// Mitsubishi GX Works2 project: EX2 (3)   PLC: FX3G

// global labels: Global1
VAR_GLOBAL
  Emergency AT X005 : BOOL;
  End_Day AT M1 : BOOL;
  Start_Day AT X007 : BOOL;
  Work_Active AT M0 : BOOL;
  Work_Light AT Y007 : BOOL;
  No_Stock AT M6 : BOOL;
  Start_Process AT X001 : BOOL;
  Analog_Input_1 AT D8280 : INT;
  Sample_Done AT M2 : BOOL;
  Regular_Type AT M3 : BOOL;
  Premium_Type AT M4 : BOOL;
  Reg_Raspberry_OK AT M20 : BOOL;
  Reg_Lemon_OK AT M21 : BOOL;
  Reg_Stabilizer_OK AT M22 : BOOL;
  Reg_Gummies_OK AT M23 : BOOL;
  Regular_Stock_OK AT M14 : BOOL;
  Prem_Raspberry_OK AT M24 : BOOL;
  Prem_Lemon_OK AT M25 : BOOL;
  Prem_Stabilizer_OK AT M26 : BOOL;
  Prem_Gummies_OK AT M27 : BOOL;
  Premium_Stock_OK AT M15 : BOOL;
  Stock_OK AT M5 : BOOL;
  Prep_Active AT M7 : BOOL;
  Prep_Timer AT TC0 : BOOL;
  Prep_Timer_Done AT TS0 : BOOL;
  Prep_Light AT Y000 : BOOL;
  Prep_Done AT M8 : BOOL;
  Start_Cooling AT X002 : BOOL;
  Cooling_Active AT M9 : BOOL;
  Cooling_Timer AT TC1 : BOOL;
  Cooling_done AT M10 : BOOL;
  Cooling_Light AT Y002 : BOOL;
  Cooling_Timer_Done AT TS1 : BOOL;
  Temp_Sensor AT X003 : BOOL;
  Mixing_Active AT M11 : BOOL;
  Mixing_Timer_Reg AT TC2 : BOOL;
  Mixing_Timer_Prem AT TC3 : BOOL;
  Blink_Timer_Done_2 AT TS5 : BOOL;
  Blink_Timer_2_Done AT TS5 : BOOL;
  Blink_Timer_1 AT TC4 : BOOL;
  Blink_Timer_1_Done AT TS4 : BOOL;
  Blink_Timer_2 AT TC5 : BOOL;
  Mixing_Light_1 AT Y005 : BOOL;
  Mixing_Light_2 AT Y006 : BOOL;
  Blink_Light_1 AT Y005 : BOOL;
  Blink_Light_2 AT Y006 : BOOL;
  Mixing_Timer_Reg_Done AT TS2 : BOOL;
  Mixing_Timer_Prem_Done AT TS3 : BOOL;
  Mixing_Done AT M12 : BOOL;
END_VAR
VAR_GLOBAL CONSTANT
  One_Package : REAL := 1.0;
END_VAR
VAR_GLOBAL
  Cycle_Reset AT M13 : BOOL;
END_VAR
VAR_GLOBAL CONSTANT
  Ten : REAL;
END_VAR
VAR_GLOBAL
  Analog_Display_Value AT D1280 : REAL;
  Analog_Output AT D8282 : INT;
  Zero AT D0 : REAL;
  Analog_Value AT D1100 : REAL;
END_VAR
VAR_GLOBAL CONSTANT
  Regular_Max : REAL;
  Premium_Min : REAL;
END_VAR
VAR_GLOBAL
  Raspberry_Stock AT D1110 : REAL;
  Reg_Raspberry_Need AT D1190 : REAL;
  Lemon_Stock AT D1120 : REAL;
  Reg_Lemon_Need AT D1200 : REAL;
  Gummies_Stock AT D1140 : REAL;
  Prem_Raspberry_Need AT D1230 : REAL;
  Prem_Lemon_Need AT D1240 : REAL;
  Storage_Count AT D1270 : REAL;
  Reg_Gummies_Need AT D1220 : REAL;
  Prem_Gummies_Need AT D1260 : REAL;
  Reg_Stabilizer_Need AT D1210 : REAL;
  Stabilizer_Stock AT D1130 : REAL;
  Prem_Stabilizer_Need AT D1250 : REAL;
  Raspberry_Need AT D1190 : REAL;
  Lemon_Need AT D1200 : REAL;
  Gummies_Need AT D1220 : REAL;
  Stabilizer_Need AT D1210 : REAL;
  Raspberry_OK AT M20 : BOOL;
  Lemon_OK AT M21 : BOOL;
  Stabilizer_OK AT M22 : BOOL;
  Gummies_OK AT M23 : BOOL;
  Input_Raspberry_Stock AT D1500 : REAL;
  Input_Lemon_Stock AT D1510 : REAL;
  Input_Stabilizer_Stock AT D1520 : REAL;
  Input_Gummies_Stock AT D1530 : REAL;
  Raspberry_Cooling_Tank AT D1300 : REAL;
  Lemon_Cooling_Tank AT D1310 : REAL;
  Mixing_Tank AT D1320 : REAL;
  Not_valid_value AT M28 : BOOL;
  Premium_Min_Check AT M29 : BOOL;
  Premium_Max_Check AT M30 : BOOL;
  Invalid_Min_Check AT M31 : BOOL;
  Invalid_Max_Check AT M32 : BOOL;
  Invalid_Range_Check AT M33 : BOOL;
  Above_10_Check AT M34 : BOOL;
END_VAR
VAR_GLOBAL CONSTANT
  Con2400 : REAL := 2400;
  Con4000 : REAL := 4000.0;
  Con_40 : REAL := 40.0;
END_VAR
VAR_GLOBAL
  Storage_multi_40 AT D1290 : REAL;
END_VAR
VAR_GLOBAL CONSTANT
  Con_210 : REAL := 210.0;
END_VAR

// task Task_01 (event TRUE, interval 0, priority 31): POU_01

PROGRAM POU_01
(* structured ladder/FBD written out as ST: instructions are called as NAME(EN, inputs, outputs); _pN, _eN, _tN stand for wires *)
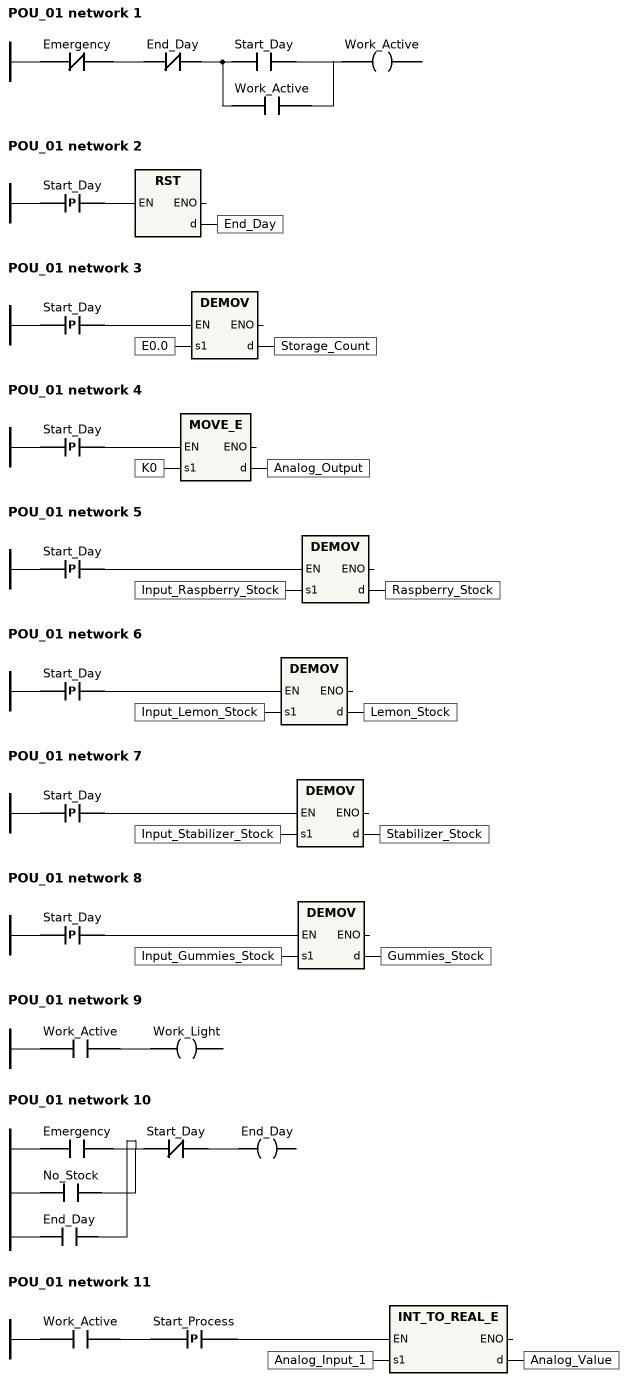
(* network 1 *)
_p1 := NOT Emergency AND NOT End_Day;
Work_Active := (_p1 AND Start_Day) OR (_p1 AND Work_Active);
(* network 2 *)
RST(LDP(TRUE, Start_Day), End_Day);
(* network 3 *)
DEMOV(LDP(TRUE, Start_Day), E0.0, Storage_Count);
(* network 4 *)
MOVE_E(LDP(TRUE, Start_Day), K0, Analog_Output);
(* network 5 *)
DEMOV(LDP(TRUE, Start_Day), Input_Raspberry_Stock, Raspberry_Stock);
(* network 6 *)
DEMOV(LDP(TRUE, Start_Day), Input_Lemon_Stock, Lemon_Stock);
(* network 7 *)
DEMOV(LDP(TRUE, Start_Day), Input_Stabilizer_Stock, Stabilizer_Stock);
(* network 8 *)
DEMOV(LDP(TRUE, Start_Day), Input_Gummies_Stock, Gummies_Stock);
(* network 9 *)
Work_Light := Work_Active;
(* network 10 *)
End_Day := (Emergency OR No_Stock OR End_Day) AND NOT Start_Day;
(* network 11 *)
INT_TO_REAL_E(Work_Active AND LDP(TRUE, Start_Process), Analog_Input_1, Analog_Value);
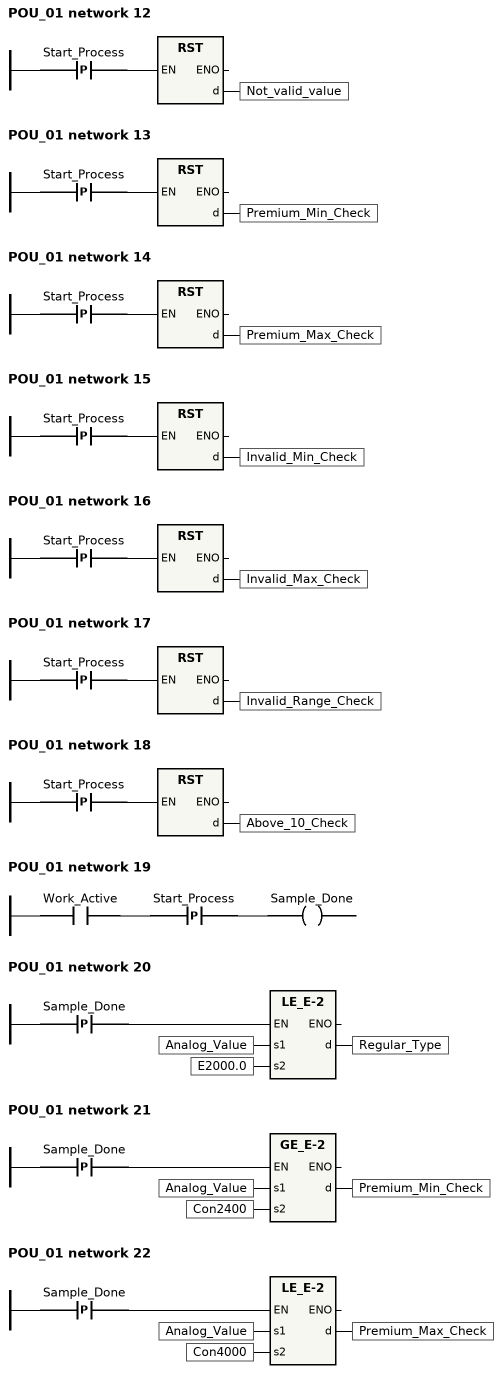
(* network 12 *)
RST(LDP(TRUE, Start_Process), Not_valid_value);
(* network 13 *)
RST(LDP(TRUE, Start_Process), Premium_Min_Check);
(* network 14 *)
RST(LDP(TRUE, Start_Process), Premium_Max_Check);
(* network 15 *)
RST(LDP(TRUE, Start_Process), Invalid_Min_Check);
(* network 16 *)
RST(LDP(TRUE, Start_Process), Invalid_Max_Check);
(* network 17 *)
RST(LDP(TRUE, Start_Process), Invalid_Range_Check);
(* network 18 *)
RST(LDP(TRUE, Start_Process), Above_10_Check);
(* network 19 *)
Sample_Done := Work_Active AND LDP(TRUE, Start_Process);
(* network 20 *)
LE_E(LDP(TRUE, Sample_Done), Analog_Value, E2000.0, Regular_Type);
(* network 21 *)
GE_E(LDP(TRUE, Sample_Done), Analog_Value, Con2400, Premium_Min_Check);
(* network 22 *)
LE_E(LDP(TRUE, Sample_Done), Analog_Value, Con4000, Premium_Max_Check);
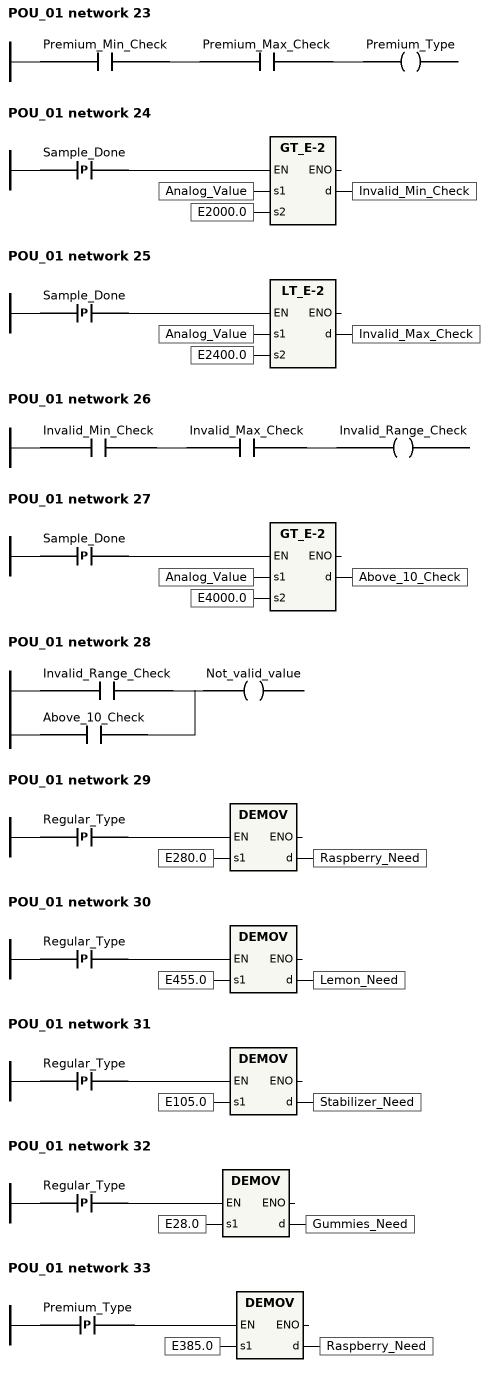
(* network 23 *)
Premium_Type := Premium_Min_Check AND Premium_Max_Check;
(* network 24 *)
GT_E(LDP(TRUE, Sample_Done), Analog_Value, E2000.0, Invalid_Min_Check);
(* network 25 *)
LT_E(LDP(TRUE, Sample_Done), Analog_Value, E2400.0, Invalid_Max_Check);
(* network 26 *)
Invalid_Range_Check := Invalid_Min_Check AND Invalid_Max_Check;
(* network 27 *)
GT_E(LDP(TRUE, Sample_Done), Analog_Value, E4000.0, Above_10_Check);
(* network 28 *)
Not_valid_value := Invalid_Range_Check OR Above_10_Check;
(* network 29 *)
DEMOV(LDP(TRUE, Regular_Type), E280.0, Raspberry_Need);
(* network 30 *)
DEMOV(LDP(TRUE, Regular_Type), E455.0, Lemon_Need);
(* network 31 *)
DEMOV(LDP(TRUE, Regular_Type), E105.0, Stabilizer_Need);
(* network 32 *)
DEMOV(LDP(TRUE, Regular_Type), E28.0, Gummies_Need);
(* network 33 *)
DEMOV(LDP(TRUE, Premium_Type), E385.0, Raspberry_Need);
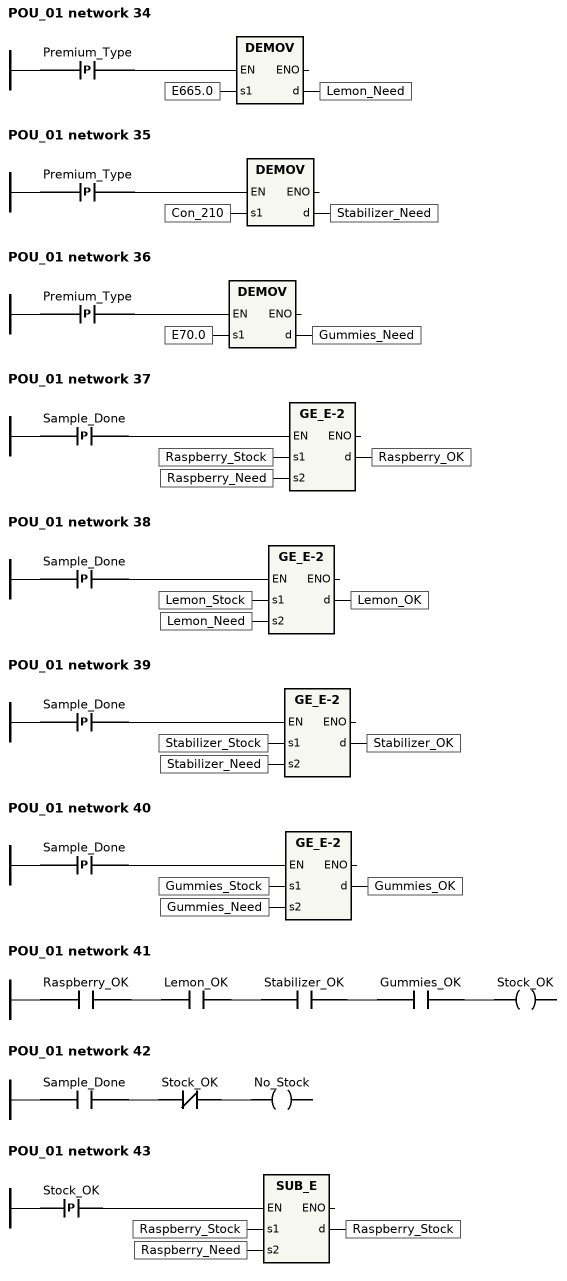
(* network 34 *)
DEMOV(LDP(TRUE, Premium_Type), E665.0, Lemon_Need);
(* network 35 *)
DEMOV(LDP(TRUE, Premium_Type), Con_210, Stabilizer_Need);
(* network 36 *)
DEMOV(LDP(TRUE, Premium_Type), E70.0, Gummies_Need);
(* network 37 *)
GE_E(LDP(TRUE, Sample_Done), Raspberry_Stock, Raspberry_Need, Raspberry_OK);
(* network 38 *)
GE_E(LDP(TRUE, Sample_Done), Lemon_Stock, Lemon_Need, Lemon_OK);
(* network 39 *)
GE_E(LDP(TRUE, Sample_Done), Stabilizer_Stock, Stabilizer_Need, Stabilizer_OK);
(* network 40 *)
GE_E(LDP(TRUE, Sample_Done), Gummies_Stock, Gummies_Need, Gummies_OK);
(* network 41 *)
Stock_OK := Raspberry_OK AND Lemon_OK AND Stabilizer_OK AND Gummies_OK;
(* network 42 *)
No_Stock := Sample_Done AND NOT Stock_OK;
(* network 43 *)
SUB_E(LDP(TRUE, Stock_OK), Raspberry_Stock, Raspberry_Need, Raspberry_Stock);
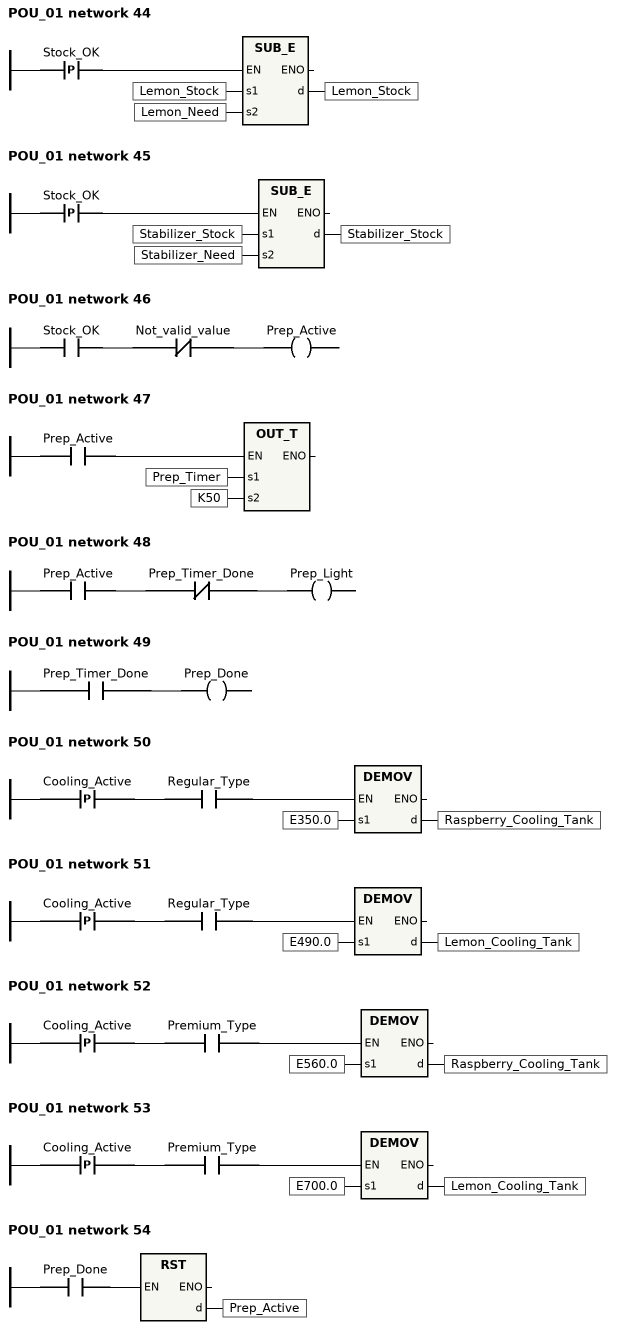
(* network 44 *)
SUB_E(LDP(TRUE, Stock_OK), Lemon_Stock, Lemon_Need, Lemon_Stock);
(* network 45 *)
SUB_E(LDP(TRUE, Stock_OK), Stabilizer_Stock, Stabilizer_Need, Stabilizer_Stock);
(* network 46 *)
Prep_Active := Stock_OK AND NOT Not_valid_value;
(* network 47 *)
OUT_T(Prep_Active, Prep_Timer, K50);
(* network 48 *)
Prep_Light := Prep_Active AND NOT Prep_Timer_Done;
(* network 49 *)
Prep_Done := Prep_Timer_Done;
(* network 50 *)
DEMOV(LDP(TRUE, Cooling_Active) AND Regular_Type, E350.0, Raspberry_Cooling_Tank);
(* network 51 *)
DEMOV(LDP(TRUE, Cooling_Active) AND Regular_Type, E490.0, Lemon_Cooling_Tank);
(* network 52 *)
DEMOV(LDP(TRUE, Cooling_Active) AND Premium_Type, E560.0, Raspberry_Cooling_Tank);
(* network 53 *)
DEMOV(LDP(TRUE, Cooling_Active) AND Premium_Type, E700.0, Lemon_Cooling_Tank);
(* network 54 *)
RST(Prep_Done, Prep_Active);
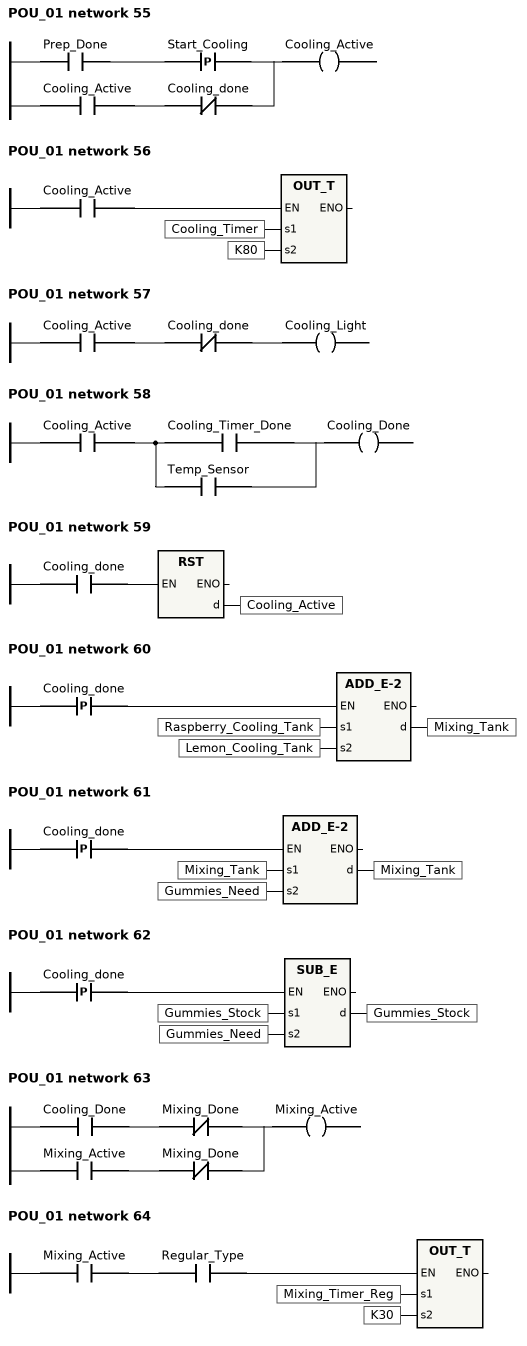
(* network 55 *)
Cooling_Active := (Prep_Done AND LDP(TRUE, Start_Cooling)) OR (Cooling_Active AND NOT Cooling_done);
(* network 56 *)
OUT_T(Cooling_Active, Cooling_Timer, K80);
(* network 57 *)
Cooling_Light := Cooling_Active AND NOT Cooling_done;
(* network 58 *)
Cooling_Done := (Cooling_Active AND Cooling_Timer_Done) OR (Cooling_Active AND Temp_Sensor);
(* network 59 *)
RST(Cooling_done, Cooling_Active);
(* network 60 *)
ADD_E(LDP(TRUE, Cooling_done), Raspberry_Cooling_Tank, Lemon_Cooling_Tank, Mixing_Tank);
(* network 61 *)
ADD_E(LDP(TRUE, Cooling_done), Mixing_Tank, Gummies_Need, Mixing_Tank);
(* network 62 *)
SUB_E(LDP(TRUE, Cooling_done), Gummies_Stock, Gummies_Need, Gummies_Stock);
(* network 63 *)
Mixing_Active := (Cooling_Done AND NOT Mixing_Done) OR (Mixing_Active AND NOT Mixing_Done);
(* network 64 *)
OUT_T(Mixing_Active AND Regular_Type, Mixing_Timer_Reg, K30);
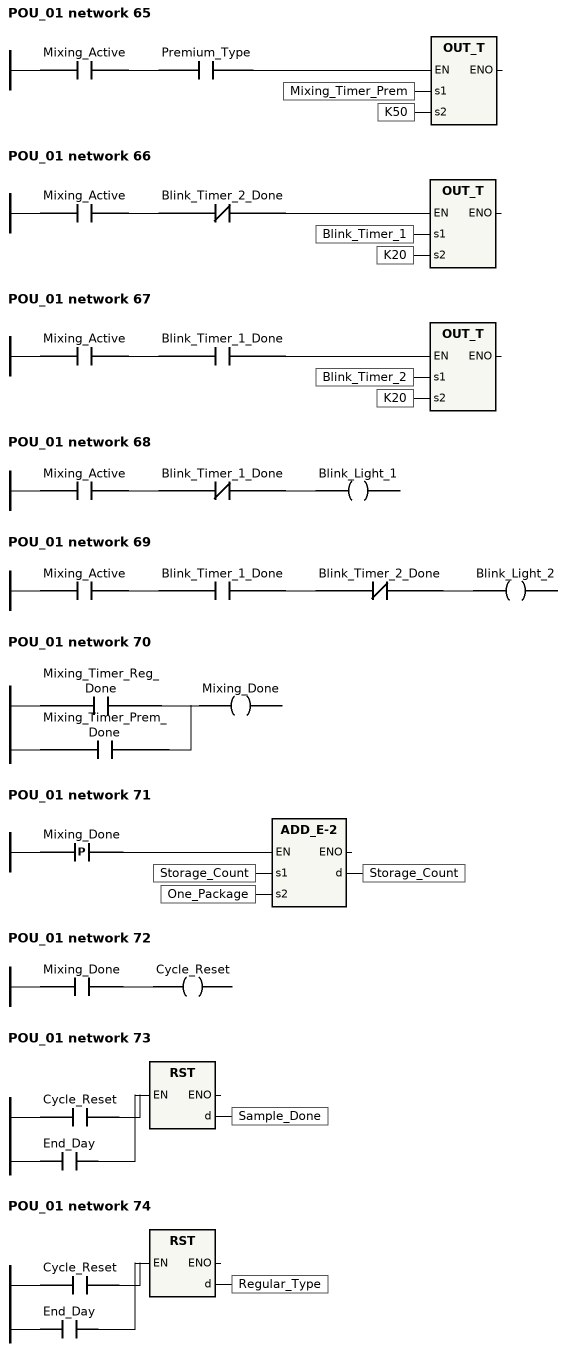
(* network 65 *)
OUT_T(Mixing_Active AND Premium_Type, Mixing_Timer_Prem, K50);
(* network 66 *)
OUT_T(Mixing_Active AND NOT Blink_Timer_2_Done, Blink_Timer_1, K20);
(* network 67 *)
OUT_T(Mixing_Active AND Blink_Timer_1_Done, Blink_Timer_2, K20);
(* network 68 *)
Blink_Light_1 := Mixing_Active AND NOT Blink_Timer_1_Done;
(* network 69 *)
Blink_Light_2 := Mixing_Active AND Blink_Timer_1_Done AND NOT Blink_Timer_2_Done;
(* network 70 *)
Mixing_Done := Mixing_Timer_Reg_Done OR Mixing_Timer_Prem_Done;
(* network 71 *)
ADD_E(LDP(TRUE, Mixing_Done), Storage_Count, One_Package, Storage_Count);
(* network 72 *)
Cycle_Reset := Mixing_Done;
(* network 73 *)
RST(Cycle_Reset OR End_Day, Sample_Done);
(* network 74 *)
RST(Cycle_Reset OR End_Day, Regular_Type);
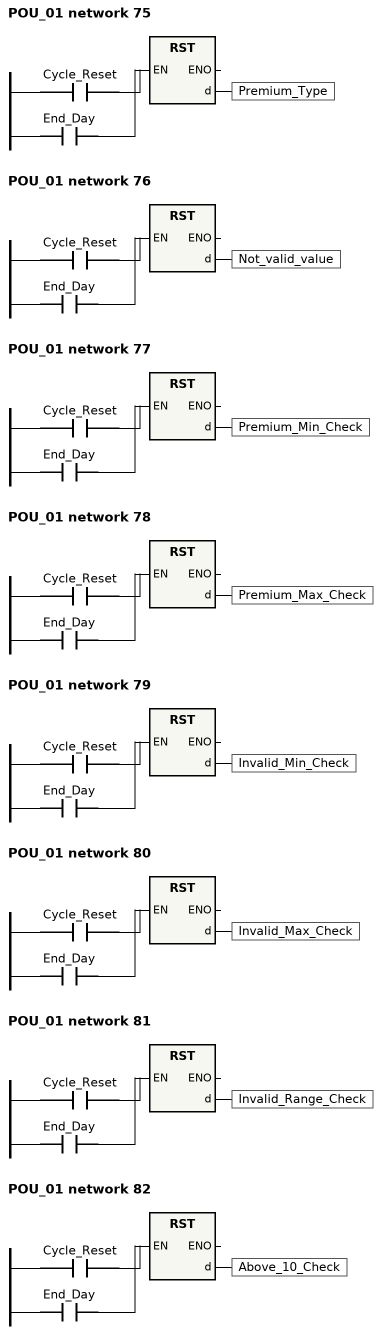
(* network 75 *)
RST(Cycle_Reset OR End_Day, Premium_Type);
(* network 76 *)
RST(Cycle_Reset OR End_Day, Not_valid_value);
(* network 77 *)
RST(Cycle_Reset OR End_Day, Premium_Min_Check);
(* network 78 *)
RST(Cycle_Reset OR End_Day, Premium_Max_Check);
(* network 79 *)
RST(Cycle_Reset OR End_Day, Invalid_Min_Check);
(* network 80 *)
RST(Cycle_Reset OR End_Day, Invalid_Max_Check);
(* network 81 *)
RST(Cycle_Reset OR End_Day, Invalid_Range_Check);
(* network 82 *)
RST(Cycle_Reset OR End_Day, Above_10_Check);
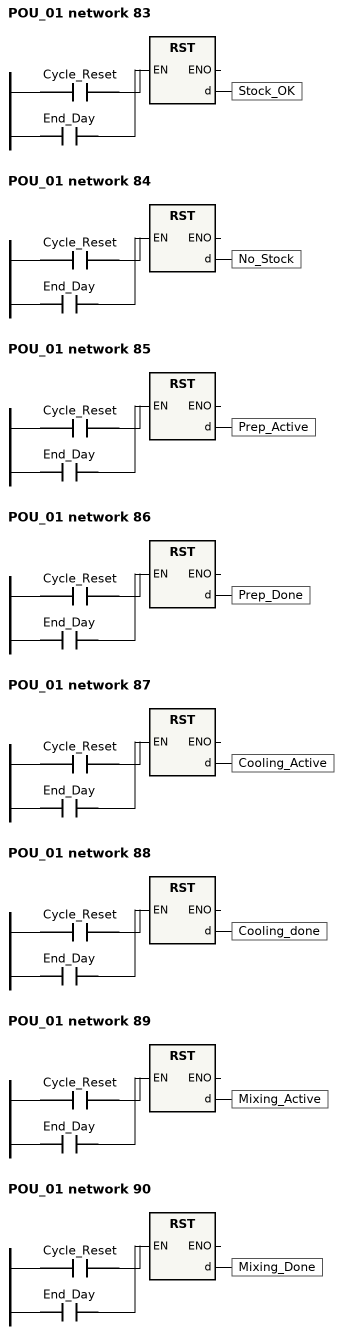
(* network 83 *)
RST(Cycle_Reset OR End_Day, Stock_OK);
(* network 84 *)
RST(Cycle_Reset OR End_Day, No_Stock);
(* network 85 *)
RST(Cycle_Reset OR End_Day, Prep_Active);
(* network 86 *)
RST(Cycle_Reset OR End_Day, Prep_Done);
(* network 87 *)
RST(Cycle_Reset OR End_Day, Cooling_Active);
(* network 88 *)
RST(Cycle_Reset OR End_Day, Cooling_done);
(* network 89 *)
RST(Cycle_Reset OR End_Day, Mixing_Active);
(* network 90 *)
RST(Cycle_Reset OR End_Day, Mixing_Done);
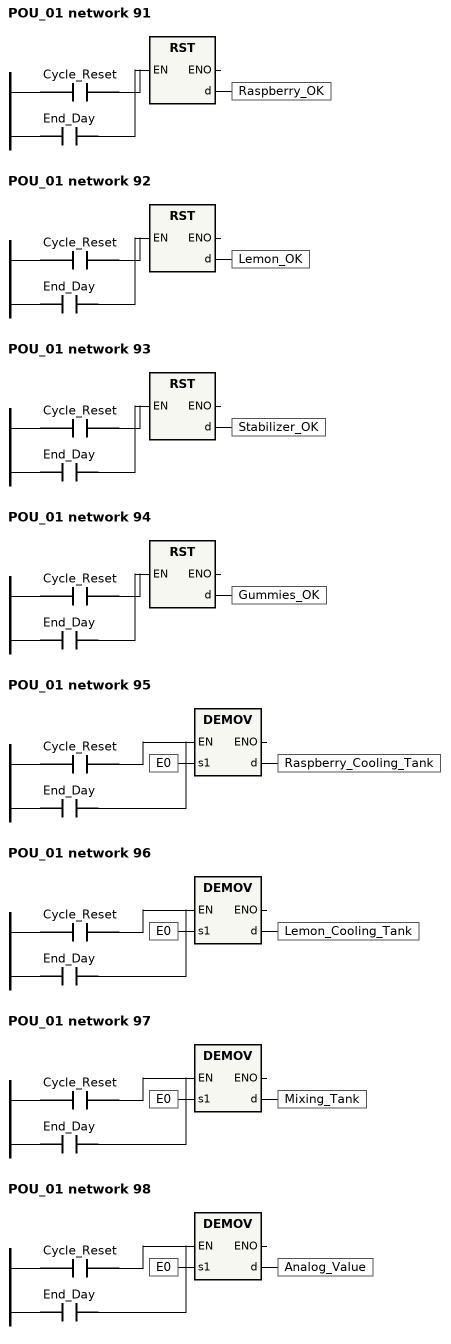
(* network 91 *)
RST(Cycle_Reset OR End_Day, Raspberry_OK);
(* network 92 *)
RST(Cycle_Reset OR End_Day, Lemon_OK);
(* network 93 *)
RST(Cycle_Reset OR End_Day, Stabilizer_OK);
(* network 94 *)
RST(Cycle_Reset OR End_Day, Gummies_OK);
(* network 95 *)
DEMOV(Cycle_Reset OR End_Day, E0, Raspberry_Cooling_Tank);
(* network 96 *)
DEMOV(Cycle_Reset OR End_Day, E0, Lemon_Cooling_Tank);
(* network 97 *)
DEMOV(Cycle_Reset OR End_Day, E0, Mixing_Tank);
(* network 98 *)
DEMOV(Cycle_Reset OR End_Day, E0, Analog_Value);
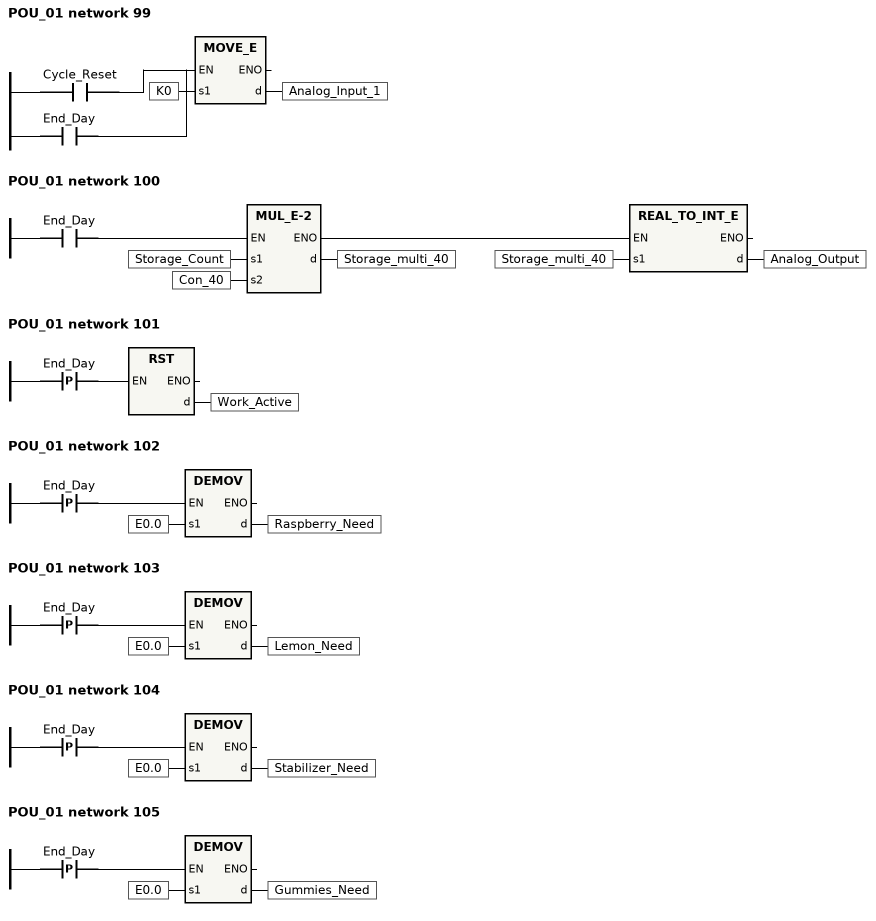
(* network 99 *)
MOVE_E(Cycle_Reset OR End_Day, K0, Analog_Input_1);
(* network 100 *)
_e1 := MUL_E(End_Day, Storage_Count, Con_40, Storage_multi_40);
REAL_TO_INT_E(_e1, Storage_multi_40, Analog_Output);
(* network 101 *)
RST(LDP(TRUE, End_Day), Work_Active);
(* network 102 *)
DEMOV(LDP(TRUE, End_Day), E0.0, Raspberry_Need);
(* network 103 *)
DEMOV(LDP(TRUE, End_Day), E0.0, Lemon_Need);
(* network 104 *)
DEMOV(LDP(TRUE, End_Day), E0.0, Stabilizer_Need);
(* network 105 *)
DEMOV(LDP(TRUE, End_Day), E0.0, Gummies_Need);
END_PROGRAM
